// TIA Portal V16 export
// export: Created 2021-07-21T13:08:43.6623794Z, ExportSetting WithDefaults, DisplayName Totally Integrated Automation Portal, DisplayVersion V16 Update 3, DisplayName TIA Portal Version Control Interface, DisplayVersion V16 Update 2, DisplayName TIA Portal Openness, DisplayVersion V16 Update 3, DisplayName STEP 7 Professional, DisplayVersion V16 Update 3, DisplayName STEP 7 Safety, DisplayVersion V16, DisplayName WinCC Professional, DisplayVersion V16 Update 3
TYPE "UT11001_St_DevValveIsol"
TITLE = Static UDT [Instrumentation] — Analog Instrument Read, Scale and Monitor
// Analogue Instrument Read and Scale
// stored: IsFailsafeCompliant false
   STRUCT
      revInfo { ExternalWritable := 'False'} : "UT01000_St_SysRevision";   // Revision information
      ___________0010_0 { ExternalAccessible := 'False'; ExternalVisible := 'False'; ExternalWritable := 'False'} : Int;
      ___________0010_1 { ExternalAccessible := 'False'; ExternalVisible := 'False'; ExternalWritable := 'False'} : Int;   // ▀▀▀▀ INSTRUMENT CONFIGURATION
      CONFIG_NO_NC : Bool;   // CONFIG — Normally open or normally closed valve (1 = normally open, 0 = normally closed)
      CONFIG_FBK_OPEN_EN : Bool;   // CONFIG — Open feedback is enabled (1 = open feedback present, 0 = no open feedback)
      CONFIG_FBK_CLOSED_EN : Bool;   // CONFIG — Closed feedback is enabled (1 = closed feedback present, 0 = no closed feedback)
      CONFIG_ESTOP_DIS : Bool;   // CONFIG — E_STOP signal disabled (1 = E_STOP not used, 0 = E_STOP in use)
      CONFIG_TRIP_DIS : Bool;   // CONFIG — TRIP signal disabled (1 = TRIP not used, 0 = TRIP in use)
      CONFIG_ILOCK_DIS : Bool;   // CONFIG — INTERLOCK signal disabled (1 = INTERLOCK not used, 0 = INTERLOCK in use)
      CONFIG_PERM_DIS : Bool;   // CONFIG — PERMISSIVE signal disabled (1 = PERMISSIVE not used, 0 = PERMISSIVE in use)
      CONFIG_TRIP_OP_CL : Bool;   // CONFIG — TRIP state (1 = open if tripped, 0 = close if tripped)
      CONFIG_ILOCK_OP_CL : Bool;   // CONFIG — INTERLOCK state (1 = open if interlocked, 0 = close if interlocked)
      CONFIG_PERM_OP_CL : Bool;   // CONFIG — PERMISSIVE permitted state (1 = permitted state open, 0 = permitted state closed)
      CONFIG_FP_DIS { ExternalWritable := 'False'; S7_SetPoint := 'True'} : Bool;   // CONFIG — Faceplate is disabled (1 = no Faceplate, 0 = normal)
      CONFIG_MAN_DIS : Bool;   // CONFIG — Manual mode is disabled (1 = no manual mode – auto only, 0 = normal)
      CONFIG_BYPASS_DIS : Bool;   // CONFIG — Bypass mode is disabled (1 = no Bypass, 0 = normal)
      CONFIG_SIM_DIS { ExternalWritable := 'False'; S7_SetPoint := 'True'} : Bool;   // CONFIG — Simulation mode is disabled (1 = no Simulation, 0 = normal)
      CONFIG_RL_EN { ExternalWritable := 'False'; S7_SetPoint := 'True'} : Bool;   // CONFIG — Remote/local mode enabled (1 = remote/local permitted, 0 = remote/local N/A)
      ___________0020_0 { ExternalAccessible := 'False'; ExternalVisible := 'False'; ExternalWritable := 'False'} : Int;
      ___________0020_1 { ExternalAccessible := 'False'; ExternalVisible := 'False'; ExternalWritable := 'False'} : Int;   // ▀▀▀▀ INSTRUMENT INFORMATION (TAG & UNITS)
      INFO_TAG { ExternalWritable := 'False'; S7_SetPoint := 'True'} : String[20];   // INFORMATION — Instrument ID tag
      ___________0030_0 { ExternalAccessible := 'False'; ExternalVisible := 'False'; ExternalWritable := 'False'} : Int;
      ___________0030_1 { ExternalAccessible := 'False'; ExternalVisible := 'False'; ExternalWritable := 'False'} : Int;   // ▀▀▀▀ INSTRUMENT TIMER DEFAULT VALUES
      TIME_OPENING_MAX { ExternalWritable := 'False'; S7_SetPoint := 'True'} : Real;   // TIMER — Initial value of opening operation timer [seconds], counts down from this value
      TIME_CLOSING_MAX { ExternalWritable := 'False'; S7_SetPoint := 'True'} : Real;   // TIMER — Initial value of closing operation timer [seconds], counts down from this value
      TIME_FBK_OPEN_SIM { ExternalWritable := 'False'; S7_SetPoint := 'True'} : Real;   // TIMER — Percentage of opening timer to expired before simulating open feedback [percentage]
      TIME_FBK_CLOSED_SIM { ExternalWritable := 'False'; S7_SetPoint := 'True'} : Real;   // TIMER — Percentage of closing timer to expired before simulating closed feedback [percentage]
   END_STRUCT;
   // revInfo.REV_BLOCK := 'UT11001';
   // revInfo.REV_NUMBER := '000.102';
   // revInfo.REV_DATE := '2021-07-21';
   // revInfo.REV_AUTHOR := 'M. Gledhill';
END_TYPE
